Staubli VAL3: onF8Event.pgx

program onF8Event()
  local bool l_bUndo
  local num l_nResult
  local string l_sNew
  local string l_sMessage
begin
  if bButton[7]
    // new one
    call alreadyExist(l_sNew,l_bUndo)
    if !l_bUndo and l_sNew!=""
      call set:new(l_sNew,l_nResult)
      if l_nResult==0
          set:bWizard=true
        if save:nBoxType==1
          call Wizard_smlBox(l_sNew,l_nResult)
        elseIf save:nBoxType==2
          call set:editBigData(l_sNew,l_nResult)
        endIf
        ///////////////////////////////////
        if l_nResult==0
          call language2:message(l_sMessage,4)
          call use:timerDialog(l_sMessage,0)
          call set:onSave()
          sEvent=l_sNew
          call buildList()
        else
           call set:delete(l_sNew,l_nResult)
           call set:onSave()
       endIf
      endIf
    endIf
  endIf
end
